FUNCTION F_ChkSettingLimit : BOOL
VAR_INPUT
	nValue		: INT;
	fValue		: LREAL;
END_VAR
VAR_IN_OUT
	stSetting 	: ST_Data_Item;
END_VAR
VAR_OUTPUT
	stInfo 		: ST_Text;
END_VAR

CASE stSetting.eDataType OF
	E_DataType.eDataType_int,
	E_DataType.eDataType_time_ms:
		F_ChkSettingLimit := F_ChkSettingLimitN(nValue, stSetting, stInfo => stInfo);
ELSE
		F_ChkSettingLimit := F_ChkSettingLimitF(fValue, stSetting, stInfo => stInfo);
END_CASE

END_FUNCTION

(* stored: Version 1.1.0.1, ProductVersion 3.1.4024.12
   POU F_ChkSettingLimit: Id {63b09c62-063e-4425-9d42-3b7500743b4c}, SpecialFunc None *)
